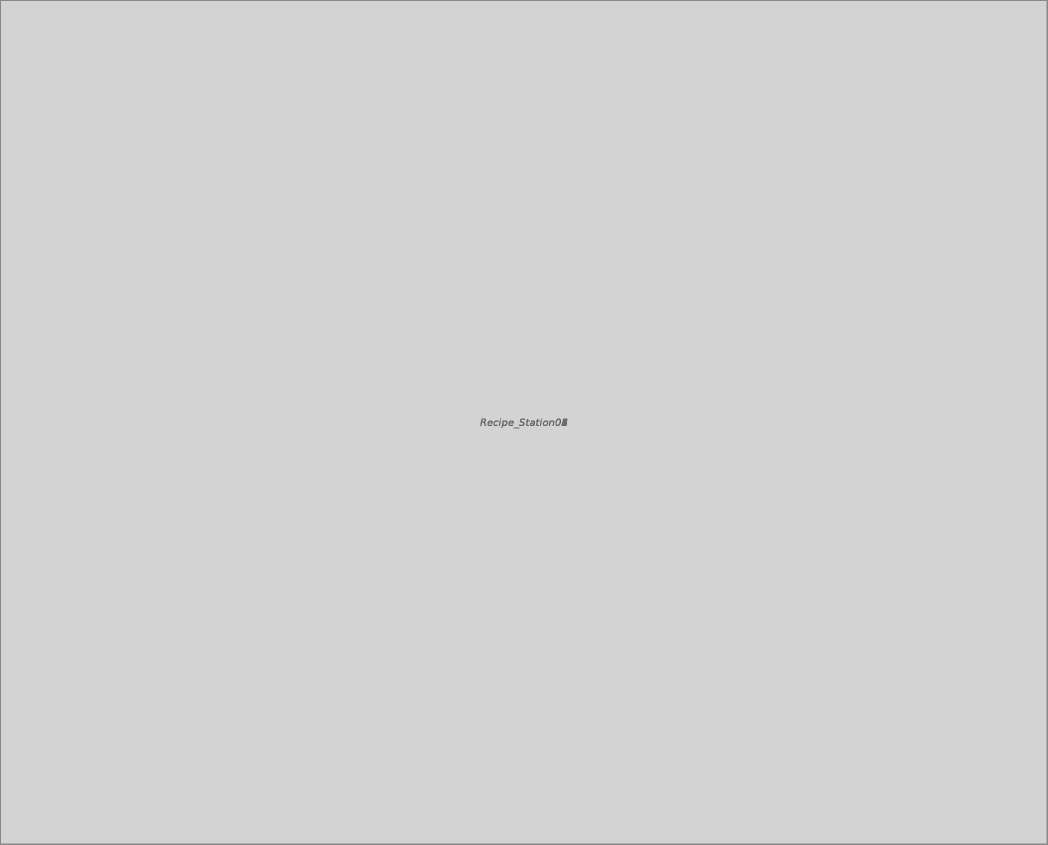
VISUALIZATION Recipe_AllStation_SSUR  // 1048x845
    Group (0,0 1048x845)
        Frame (0,0 1048x845), invisible if: iStationNo<>1
            shows Recipe_Station01()
        Frame (0,0 1048x845), colour toggle: iStationNo<>2
            shows Recipe_Station02()
        Frame (0,0 1048x845), invisible if: iStationNo<>3
            shows Recipe_Station03()
        Frame (0,0 1048x845), invisible if: iStationNo<>4
            shows Recipe_Station04()
        Frame (0,0 1048x845), invisible if: iStationNo<>5
            shows Recipe_Station05()
        Frame (0,0 1048x845), invisible if: iStationNo<>6
            shows Recipe_Station06()
END_VISUALIZATION

(* stored: Version 1.1.0.1, ProductVersion 3.1.4024.12
   Visu Recipe_AllStation_SSUR: Id {5f956e09-528e-45b9-9b12-9cea0aea383b} *)
